{attribute 'qualified_only'}
VAR_GLOBAL CONSTANT
	iParamList : INT := 1;
END_VAR

(* stored: Version 1.1.0.1, ProductVersion 3.1.4022.18
   GVL ParameterList: Id {0b0db9fe-bb0d-485d-ac11-72d56aa6fb3e}, ParameterList True *)
